(* IEC 61131-3 sources: plcassist-cli/packages/volt-lsp-iec/test-corpus/bakon-nano/Device/Plc Logic/Application/POUs/LenzeFunctions/KinematicTransformations, 4 files *)

(* ---- L_MKT_StopErrorKinematic.fb ---- *)
FUNCTION_BLOCK L_MKT_StopErrorKinematic
VAR_INPUT
	xEnable						: BOOL;
	scPosition_InverseKinematic : L_MMB_PositionValue;
	xError_InverseKinematic		: BOOL;					(* xError OutPut inverse Kinematik									*)
	wErrorID_InverseKinematic	: WORD;					(* wErrorId Output inverse Kinematik								*)
	lfStopDeceleration			: LREAL;				(* MC_Stop:		Deceleration										*)
END_VAR
VAR_OUTPUT
	xError						: BOOL;
	xAborted					: BOOL;
	xMC_Stop					: BOOL;
	xMC_StopDone				: BOOL;
END_VAR
VAR_IN_OUT
	Axis_VIRTUAL_X				: AXIS_REF;
	Axis_VIRTUAL_Y				: AXIS_REF;
END_VAR

VAR
	sToDo					: STRING;
	sErrorID				: STRING;
	MC_Stop_X_FB			: MC_Stop;
	MC_Stop_Y_FB			: MC_Stop;
	scPositionError			: L_MMB_PositionValue;
	R_TRIG_xEnable			: R_TRIG;

	byStepper				: BYTE:=0;
END_VAR

(****************************************************************************************************************)
(* INITIALISIRUNG FB																							*)
(****************************************************************************************************************)
	R_TRIG_xEnable(CLK:=xEnable , Q=> );
	(********************************************)
	(* MC_stop									*)
	(********************************************)
	MC_Stop_X_FB(Execute:=xMC_Stop, Deceleration:= lfStopDeceleration, Axis:=Axis_VIRTUAL_X );
	MC_Stop_Y_FB(Execute:=xMC_Stop, Deceleration:= lfStopDeceleration, Axis:=Axis_VIRTUAL_Y );

	IF (Axis_VIRTUAL_X.eAxisState=L_MC1P_AXIS_STATE.Disabled OR MC_Stop_x_FB.Done) AND			//SMC_State was compared with 0 > power off
		(Axis_VIRTUAL_Y.eAxisState=L_MC1P_AXIS_STATE.Disabled OR MC_Stop_Y_FB.Done)  THEN
		xMC_StopDone:= TRUE;
	ELSE
		xMC_StopDone:= FALSE;
	END_IF

(********************************************)
(* INIT										*)
(********************************************)
	IF R_TRIG_xEnable.Q THEN
		xAborted:=FALSE;
		xError := FALSE;
		xMC_Stop:= FALSE;
		byStepper:=1;
	END_IF
	IF NOT(xEnable) THEN
		byStepper:=0;
	END_IF

(********************************************)
(* StateMaschine							*)
(********************************************)

	CASE byStepper OF
		0: (* Not ENABLE *)
			;

		1:(* NoError *)
			sErrorID:='NoError';
			sToDo:='Position is Ok';
			xError:=FALSE;
			(* Check the Errors *)
			IF xError_InverseKinematic THEN
				byStepper:=10;
			END_IF
			(* Check the real Axis A1,2,3 and A4 position *)
			(* EndersR: Überwachung der Riemenlänge*)
			IF scPosition_InverseKinematic.lrA1 < -100000 OR scPosition_InverseKinematic.lrA1 > 100000 THEN
				byStepper:=10;
			ELSIF scPosition_InverseKinematic.lrA2 < -100000 OR scPosition_InverseKinematic.lrA2 > 100000 THEN
				byStepper:=10;

			END_IF

		10:	xMC_Stop:=TRUE;
			xError:=TRUE;
			byStepper:=12;

		12: (* ErrorInput *)
			sErrorID:='ErrorInput';
			IF xMC_StopDone THEN
				scPositionError	:= scPosition_InverseKinematic;
				scPositionError.lrX	:= Axis_VIRTUAL_X.lrSetPosition;
				scPositionError.lrY	:= Axis_VIRTUAL_Y.lrSetPosition;
				xMC_Stop:=FALSE;
				byStepper:=14;
			END_IF
		14: (* ErrorID *)
			CASE wErrorID_InverseKinematic OF
				1000:   byStepper:=16; 	(*NoEROOR*)
				1001: 	byStepper:=70; 	(*A1-Limited*)

			END_CASE
		16:(* Check the real Axis A1,2,3 and A4 position whis Safety of Deltapos*)

				byStepper:=1;
	END_CASE

END_FUNCTION_BLOCK

(* ---- L_TK1A_DirectKinematicRoller45.fb ---- *)
(****************************************************************************************************)
(*	 L_TK1A_DirectKinematicRoller45																	*)
(****************************************************************************************************)
(*	LENZE CbA																					*)
(****************************************************************************************************)
(*	Direct Kinematic Roller-Picker Robot (2D)														*)
(*																									*)
(*	Note:																							*)
(* #1 x_E=f(q) : q roller-axes (A1,A2), x_E endeffectorpositions (X,Y)                         		*)
(* #2 Input: Jointspace (A1,A2,(A3=Q3),(A4=Q4)) 													*)
(* #3 Output: Taskspace (X, Y)																		*)
(****************************************************************************************************)
(*	Historie:																						*)
(****************************************************************************************************)

FUNCTION_BLOCK L_TK1A_DirectKinematicRoller45
VAR_INPUT
	scActPositionIn:		L_MMB_PositionValue;
	scParamRobot:			L_TK1A_ParamRobotRoller45;
	scLimitRobot:			L_TK1A_LimitsRobotRoller45;
END_VAR
VAR_OUTPUT
	scActPositionOut:		L_MMB_PositionValue;
	xError:					BOOL;
END_VAR
VAR
	lrS1							: LREAL;
	lrS2							: LREAL;
	bNEw: BOOL:=TRUE;
END_VAR

(************************************************)
(* basic configuration of the robot:			*)
(* see picture 1								*)
(* A1/A2-coordinate-system is rotated 45° ccw	*)
(* coordinate-system rotation:					*)
(* A2 = X-part of rotated system				*)
(* A1 = Y-part of rotated system				*)
(* A2 =  X*cos45° + Y*sin45°					*)
(* A1 = -X*sin45° + Y*cos45						*)
(************************************************)
IF NOT bNew THEN
lrS1 := scParamRobot.lrFeedConstantA1*scActPositionIn.lrA1/360;
lrS2 := scParamRobot.lrFeedConstantA2*scActPositionIn.lrA2/360;

scActPositionOut.lrX:= 0.5*lrS1 + 0.5*lrS2;
scActPositionOut.lrY:= 0.5*lrS1 - 0.5*lrS2;
ELSE
lrS1 :=scActPositionIn.lrA1;
lrS2 :=scActPositionIn.lrA2;

scActPositionOut.lrX:= 0.5*lrS1 + 0.5*lrS2;
scActPositionOut.lrY:= 0.5*lrS1 - 0.5*lrS2;
END_IF

(************************************************)
(************************************************)
(**  										   **)
(**  				ERRORCHEcK				   **)
(**  										   **)
(************************************************)
(************************************************)

END_FUNCTION_BLOCK

(* ---- L_TK1A_InverseKinematicRoller45.fb ---- *)
(****************************************************************************************************)
(*	 L_TK1A_InverseKinematicRoller45																	*)
(****************************************************************************************************)
(*	LENZE CbA																					*)
(****************************************************************************************************)
(*	Inverse Kinematic Roller-Picker Robot (2D)														*)
(*																									*)
(*	Note:																							*)
(* #1 q=g(x_E) : q roller-axes (A1,A2), x_E endeffectorpositions (X,Y)                         		*)
(* #2 Input: Taskspace (X, Y)																		*)
(* #3 Output: Jointspace (A1,A2,(A3=Q3),(A4=Q4))													*)
(****************************************************************************************************)
(*	Historie:																						*)

(****************************************************************************************************)

FUNCTION_BLOCK L_TK1A_InverseKinematicRoller45
VAR_INPUT
	scActPositionIn:		L_MMB_PositionValue;
	scParamRobot:			L_TK1A_ParamRobotRoller45;
	scLimitRobot:			L_TK1A_LimitsRobotRoller45;
END_VAR
VAR_OUTPUT
	scActPositionOut:		L_MMB_PositionValue;
	xError:					BOOL;
	wErrorID:				WORD;
END_VAR
VAR
	lrS1							: LREAL;
	lrS2							: LREAL;
	bNew: BOOL:=TRUE;
END_VAR

(************************************************)
(* basic configuration of the robot:			*)
(* see picture 1								*)
(* A1/A2-coordinate-system is rotated 45° ccw	*)
(* coordinate-system rotation:					*)
(* A2 = X-part of rotated system				*)
(* A1 = Y-part of rotated system				*)
(* A2 =  X*cos45° + Y*sin45°					*)
(* A1 = -X*sin45° + Y*cos45						*)
(************************************************)
IF NOT bNew THEN
lrS1	:=		  scActPositionIn.lrX +   scActPositionIn.lrY;
lrS2	:=		 scActPositionIn.lrX -  scActPositionIn.lrY;

scActPositionOut.lrA1:=lrS1*360/scParamRobot.lrFeedConstantA1;
scActPositionOut.lrA2:=lrS2*360/scParamRobot.lrFeedConstantA2;
ELSE
lrS1	:=		  scActPositionIn.lrX +   scActPositionIn.lrY;
lrS2	:=		 scActPositionIn.lrX -  scActPositionIn.lrY;

scActPositionOut.lrA1:=lrS1;
scActPositionOut.lrA2:=lrS2;
END_IF
(************************************************)
(************************************************)
(**  										   **)
(**  				ERRORCHEcK				   **)
(**  										   **)
(************************************************)
(************************************************)

END_FUNCTION_BLOCK

(* ---- Transform_XY_FrontRear.fb ---- *)
FUNCTION_BLOCK Transform_XY_FrontRear
VAR_INPUT
	xEnable							: BOOL;
	xSetRealPosToVirtualAxis		: BOOL;
	scParamRobot					:L_TK1A_ParamRobotRoller45;
	scLimitRobot					:L_TK1A_LimitsRobotRoller45;
END_VAR
VAR_IN_OUT
	Drive_X							: AXIS_REF;
	Drive_Y							: AXIS_REF;
	Drive_A1						: AXIS_REF;
	Drive_A2						: AXIS_REF;
END_VAR
VAR_OUTPUT
	xBusy							: BOOL;
	xError							: BOOL;
	xVirtualAxisPositionsSetOK		: BOOL;
	lrActPosX						: LREAL;
	lrActPosY						: LREAL;
END_VAR
VAR
	xInit							: BOOL;

	(*AxisControll*)
	MC_SetPosition_X_FB				: MC_SetPosition;
	MC_SetPosition_Y_FB				: MC_SetPosition;
	SMC_ControlAxisByPos_A1_FB 		: L_MC1P_FollowSetValues;
	SMC_ControlAxisByPos_A2_FB 		: L_MC1P_FollowSetValues;

	(*ROBOT_FB*)
	L_MKT_DirectKinematic_FB		: L_TK1A_DirectKinematicRoller45;
	L_MKT_InverseKinematic_FB		: L_TK1A_InverseKinematicRoller45;
(*	FB_Visu							: FB_VisuRoller45;*)
	L_MKT_StopErrorKinematic_FB		: L_MKT_StopErrorKinematic;
	MC_Halt_A1						: MC_Halt;
	MC_Halt_A2						: MC_Halt;

	xDriveA1Enabled					: BOOL;
	xDriveA2Enabled					: BOOL;
END_VAR

(****************************************************************************************************************)
(* INITIALISIRUNG FB																							*)
(****************************************************************************************************************)
(****************************************************************************************************************)

	(********************************************)
	(* DirectKinematic							*)
	(********************************************)
		L_MKT_DirectKinematic_FB.scActPositionIn.lrA1:=Drive_A1.lrActPosition;
		L_MKT_DirectKinematic_FB.scActPositionIn.lrA2:=Drive_A2.lrActPosition;

		L_MKT_DirectKinematic_FB(
			scActPositionIn:= ,
			scParamRobot:=scParamRobot ,
			scLimitRobot:=scLimitRobot ,
			scActPositionOut=> ,
			xError=> );

		lrActPosX := L_MKT_DirectKinematic_FB.scActPositionOut.lrX;
		lrActPosY := L_MKT_DirectKinematic_FB.scActPositionOut.lrY;

	(********************************************)
	(* InverseKinematic							*)
	(********************************************)
		L_MKT_InverseKinematic_FB.scActPositionIn.lrX := Drive_X.lrSetPosition;
		L_MKT_InverseKinematic_FB.scActPositionIn.lrY := Drive_Y.lrSetPosition;

		L_MKT_InverseKinematic_FB(
			scActPositionIn:= ,
			scParamRobot:=scParamRobot ,
			scLimitRobot:=scLimitRobot ,
			scActPositionOut=> ,
			xError=> );

	(****************************************************************************)
	(*Control_AxisByPos	A1,A2,A3	xBusy:=TRUE THEN Enable Control A1,1,2,3   *)
	(***************************************************************************)
	(********************************************)
	(* SETPositon Virtual Axis					*)
	(********************************************)
		(* MC_SetPosition_X_FB(Position:= -L_MKT_DirectKinematic_FB.scActPositionOut.lrX,  Mode:= FALSE, 	Axis:= Drive_X );*)
		MC_SetPosition_X_FB(
			Axis:= Drive_X,
			Execute:= ,
			Position:= L_MKT_DirectKinematic_FB.scActPositionOut.lrX,
			Relative:= FALSE,
			ExecutionMode:= ,
			RestartPositioning:= ,
			UseSettingsFromHomingMode:= ,
			Done=> ,
			Busy=> ,
			Error=> ,
			ErrorID=> );

		(* MC_SetPosition_Y_FB(Position:= -L_MKT_DirectKinematic_FB.scActPositionOut.lrY, Mode:= FALSE,		Axis:= Drive_Y );	*)
		MC_SetPosition_Y_FB(
			Axis:= Drive_Y,
			Execute:= ,
			Position:= L_MKT_DirectKinematic_FB.scActPositionOut.lrY,
			Relative:= FALSE,
			ExecutionMode:= ,
			RestartPositioning:= ,
			UseSettingsFromHomingMode:= ,
			Done=> ,
			Busy=> ,
			Error=> ,
			ErrorID=> );

		MC_Halt_A1(
			Execute:= ,
			Deceleration:= ,	//SET IN CODE 41 > Was fSWMaxDeceleration in old motion
			Jerk:= ,			//SET IN CODE 43
			Axis:= Drive_A1,
			Done=> ,
			CommandAborted=> ,
			Error=> ,
			ErrorID=> );

		MC_Halt_A2(
			Execute:= ,
			Deceleration:= ,	//SET IN CODE 41 > Was fSWMaxDeceleration in old motion
			Jerk:= ,			//SET IN CODE 43
			Axis:= Drive_A2,
			Done=> ,
			CommandAborted=> ,
			Error=> ,
			ErrorID=> );

		SMC_ControlAxisByPos_A1_FB(
			Axis:= Drive_A1,
			xExecute:= xBusy,
			xContinuousUpdate:= TRUE,
			lrPosition:= L_MKT_InverseKinematic_FB.scActPositionOut.lrA1,
			lrVelocity:= Drive_A1.scPar.MaxVelocity,
			lrAcceleration:= Drive_A1.scPar.MaxAcceleration,
			eSetValueMode:= L_MC1P_SetValueMode.Pos,
			xBusy=> ,
			xCommandAborted=> ,
			xError=> ,
			eErrorID=> );

		SMC_ControlAxisByPos_A2_FB(
			Axis:= Drive_A2,
			xExecute:= xBusy,
			xContinuousUpdate:= TRUE,
			lrPosition:= L_MKT_InverseKinematic_FB.scActPositionOut.lrA2,
			lrVelocity:= Drive_A2.scPar.MaxVelocity,
			lrAcceleration:= Drive_A2.scPar.MaxAcceleration,
			eSetValueMode:= L_MC1P_SetValueMode.Pos,
			xBusy=> ,
			xCommandAborted=> ,
			xError=> ,
			eErrorID=> );

	(********************************************)
	(* ERROR_STOP					*)
	(********************************************)
		L_MKT_StopErrorKinematic_FB(
			xEnable:= xBusy,
			scPosition_InverseKinematic:= L_MKT_InverseKinematic_FB.scActPositionOut,
			xError_InverseKinematic:= L_MKT_InverseKinematic_FB.xError,
			wErrorID_InverseKinematic:=L_MKT_InverseKinematic_FB.wErrorID ,
			lfStopDeceleration:= 500,
			Axis_VIRTUAL_X:= Drive_X ,
			Axis_VIRTUAL_Y:= Drive_Y,
			xError=> ,
			xMC_Stop=> ,
			xMC_StopDone=> );

		IF L_MKT_StopErrorKinematic_FB.xAborted THEN
			xBusy:= FALSE;
		END_IF

(************************************************************************************)
(* 										INIT										*)
(************************************************************************************)
(************************************************************************************)
	xDriveA1Enabled					:=Drive_A1.xAxisAvailable AND Drive_A1.xDriveEnabled;
	xDriveA2Enabled					:=Drive_A1.xAxisAvailable AND Drive_A1.xDriveEnabled;

	IF NOT xEnable THEN
		xInit 						:= FALSE;
		xVirtualAxisPositionsSetOK	:= FALSE;
		xBusy						:= FALSE;
		MC_Halt_A1.Execute			:= xDriveA1Enabled;
		MC_Halt_A2.Execute			:= xDriveA2Enabled;
		MC_SetPosition_X_FB.Execute	:= FALSE;
		MC_SetPosition_Y_FB.Execute	:= FALSE;
	ELSE
		IF xError THEN
		MC_Halt_A1.Execute			:= xDriveA1Enabled;
		MC_Halt_A2.Execute			:= xDriveA2Enabled;
		ELSE
		MC_Halt_A1.Execute			:= FALSE;
		MC_Halt_A2.Execute			:= FALSE;
		END_IF

		IF NOT xInit OR xSetRealPosToVirtualAxis THEN
			xInit 						:= TRUE;
			xSetRealPosToVirtualAxis 	:= FALSE;
			xVirtualAxisPositionsSetOK	:= FALSE;
			(********************************************)
			(* SET X,Y,Z								*)
			(********************************************)
			MC_SetPosition_X_FB.Execute:= TRUE;
			MC_SetPosition_Y_FB.Execute:= TRUE;
		END_IF
	END_IF

(************************************************************************************)
(*  	bBusy:=True (X,Y,Z are set AND NOT DirectKinematic_FB.bError)				*)
(************************************************************************************)
(************************************************************************************)
	IF MC_SetPosition_X_FB.Done AND
		MC_SetPosition_Y_FB.Done THEN

		MC_SetPosition_X_FB.Execute:= FALSE;
		MC_SetPosition_Y_FB.Execute:= FALSE;

		xVirtualAxisPositionsSetOK  := TRUE;

		IF NOT L_MKT_DirectKinematic_FB.xError THEN
			xBusy 					:=TRUE;
		END_IF
	END_IF

(************************************************************************************)
(************************************************************************************)
(* 								Error 												*)
(************************************************************************************)
(************************************************************************************)
	IF L_MKT_InverseKinematic_FB.xError OR
		L_MKT_DirectKinematic_FB.xError OR
		SMC_ControlAxisByPos_A1_FB.xError OR
		SMC_ControlAxisByPos_A2_FB.xError OR
		SMC_ControlAxisByPos_A1_FB.xCommandAborted OR
		SMC_ControlAxisByPos_A2_FB.xCommandAborted THEN
		xError						:=TRUE;
	ELSE
		xError						:=FALSE;
	END_IF

(************************************************************************************)
(************************************************************************************)
(* 								Visu												*)
(************************************************************************************)
(************************************************************************************)
(*
(*// Error from Direct and Invers Kinematic*)
IF L_MKT_DirectKinematic_FB.xError AND NOT(xBusy) THEN
	FB_Visu.xError:=TRUE;
	FB_Visu.wErrorID:= L_MKT_DirectKinematic_FB.wErrorID;
	ELSIF L_MKT_InverseKinematic_FB.xError AND xBusy THEN
	FB_Visu.xError:=TRUE;
	FB_Visu.wErrorID:= L_MKT_InverseKinematic_FB.wErrorID;
	ELSE
	FB_Visu.xError:=FALSE;
END_IF

	FB_Visu.scActPositionIn.lrA1:=Drive_A1.lrSetPosition;
	FB_Visu.scActPositionIn.lrA2:=Drive_A2.lrSetPosition;

	(*Virtual axes*)
	FB_Visu.scActPositionIn.lrX:=Drive_X.lrSetPosition;
	FB_Visu.scActPositionIn.lrY:=Drive_Y.lrSetPosition;
	FB_Visu.scActPositionIn.lrZ:=Drive_Z.lrSetPosition;
	FB_Visu(scActPositionIn:= , scParamRobot:= scParamRobot);
*)

END_FUNCTION_BLOCK
